// TIA Portal V19 export
TYPE "OP_Int"
   STRUCT
      O_ComActive : Bool;   // Feedback communication activ
      O_Fault : Bool;   // Fault communication
      I_DataStorage : Bool;   // activate DataStorage (only if master and device are V1.1)
      I_BlockParam : Bool;   // activate Block Parameter Setting (only if master and device are V1.1)
      IO_ReadReq : Bool;   // Request reading
      IO_WriteReq : Bool;   // Request writing
      IO_Ackn : Bool;   // Request acknowledge
      IO_ParamConfigFault : Bool;   // Read parameter configuration fault collection
   END_STRUCT;
END_TYPE
